//converts a RobotPose into a ARRAY [0..3] OF LREAL
FUNCTION RP2ARRAY : ARRAY [0..3] OF LREAL
VAR_INPUT
	pose: RobotPose;
END_VAR
VAR
END_VAR

RPS2ARRAY[0] := pose.x;
RPS2ARRAY[1] := pose.y;
RPS2ARRAY[2] := pose.theta;
RPS2ARRAY[3] := pose.e;

END_FUNCTION

(* stored: Version 1.1.0.1, ProductVersion 3.1.4024.11
   POU RP2ARRAY: Id {c71992dc-061f-4917-9525-79ee51a46dd7}, SpecialFunc None *)
